INTERFACE I_Safety

METHOD Run : BOOL
VAR_INPUT
END_VAR
END_METHOD

PROPERTY stSafety : REFERENCE TO ST_SafetyStruct
GET
END_GET
SET
END_SET
END_PROPERTY

END_INTERFACE

(* stored: Version 1.1.0.1, ProductVersion 3.1.4024.11
   Itf I_Safety: Id {2877aa5d-dc39-4451-b88e-d80e2abb8ffa}
   Method Run: Id {676a53f5-f790-48f9-bc75-81545fd166b8}
   Property stSafety: Id {f8f4336a-7009-4369-a2dd-03e68da56c08}
   Get Get: Id {411d0718-7472-477f-b424-9db778e52990}
   Set Set: Id {4186a198-fc93-4606-a2ef-6950e72727a7} *)
